(* IEC 61131-3 sources: ahu-codesys/codesys/src/motor-control, 2 files *)

(* ---- GVL_Motor.st ---- *)
{attribute 'qualified_only'}
VAR_GLOBAL
    (* Inputs - Commands from HMI *)
	StartCmd AT %QX0.0        : BOOL;
    StopCmd AT %QX0.1         : BOOL;
    ResetCmd AT %QX0.2        : BOOL;
    EStop AT %QX0.3           : BOOL;
    OverloadTrip AT %QX0.4    : BOOL;

    (* Internal *)
    MotorInternal  : BOOL;
    OverloadMem     : BOOL;

    (* Outputs - Status to HMI *)
    MotorOut AT %QX0.5     : BOOL;
    OverloadAlarm AT %QX0.6   : BOOL;

	(* Motor Start Counter *)
	StartCounter : CTU;
	MotorOutRising : R_TRIG;
END_VAR

(* ---- PLC_PRG_Motor.st ---- *)
(* Motor seal-in logic *)
GVL.MotorInternal := (GVL.StartCmd OR GVL.MotorInternal) AND NOT GVL.StopCmd AND NOT GVL.EStop;

(* Overload Latch - stays TRUE until reset *)
GVL.OverloadMem := (GVL.OverloadTrip OR GVL.OverloadMem) AND NOT GVL.ResetCmd;

(* Overload Alarm Output *)
GVL.OverloadAlarm := GVL.OverloadMem;

(* Motor output - runs only if internal seal-in is active  AND no overload AND no EStop *)
GVL.MotorOut := GVL.MotorInternal AND NOT GVL.OverloadMem AND NOT GVL.EStop;

(* If overload trips, break the seal-in *)
IF GVL.OverloadMem THEN
	GVL.MotorInternal := FALSE;
END_IF
